FUNCTION TryConvert_TIME_TO_SINT : BOOL
VAR_INPUT
	in : TIME;
	out : REFERENCE TO SINT;
END_VAR

IF in > DatatypeLimits.MAX_VALUE_OF_TIME_WHICH_CAN_BE_HELD_IN_A_SINT THEN
	RETURN;
END_IF

out := TIME_TO_SINT(in);
TryConvert_TIME_TO_SINT := TRUE;

END_FUNCTION

(* stored: Version 1.1.0.1, ProductVersion 3.1.4024.12
   POU TryConvert_TIME_TO_SINT: Id {e9239f1e-f386-44dc-9a42-5361bf870df9}, SpecialFunc None *)
